{attribute 'GeneratedUsingTerminal: EPP6228-0022-0016'}
{attribute addProperty BoxType "EPP6228-0022-0016"}
{attribute addProperty Id "AdsAddrAT %I*.TcoAmsAddr0AoeNetIdAT %I*.TcoAmsNetId0StateAT %I*UINT2"}
{attribute addProperty CRC "1103447971"}
{attribute addProperty Size "2"}
TYPE InfoData_41C547A3 :
STRUCT
	{attribute addProperty Name "AdsAddr"}
	AdsAddr AT %I* : .TcoAmsAddr;
	{attribute addProperty Name "AoeNetId"}
	AoeNetId AT %I* : .TcoAmsNetId;
	{attribute addProperty Name "State"}
	State AT %I* : UINT;
END_STRUCT
END_TYPE

(* stored: Version 1.2.0.0, ProductVersion 3.1.4024.9
   DUT InfoData_41C547A3: Id {001b2331-414e-41ce-ace2-dbe06d37e530} *)
